FUNCTION_BLOCK FB_Blinker
VAR_INPUT
	bStart: BOOL;
	tTime: TIME;
END_VAR
VAR_OUTPUT
	bOutPut: BOOL;
END_VAR
VAR
	T1: TON;
	T2: TON;
END_VAR

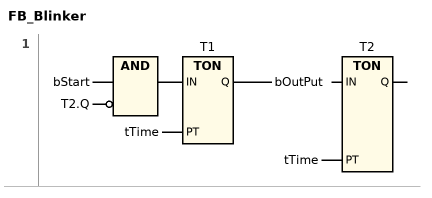
// NETWORK 1
T1(IN := bStart AND NOT T2.Q, PT := tTime); // TON
bOutPut := T1.Q;
T2(IN := T1.Q, PT := tTime); // TON

END_FUNCTION_BLOCK

(* stored: Version 1.1.0.1, ProductVersion 3.1.4024.2
   POU FB_Blinker: Id {005b9bc4-3cbc-47e7-8e03-36c999586b6a}, SpecialFunc None *)
